// TwinCAT 3 PLC project Untitled1
// ProgramVersion: 3.1.4024.0
// libraries:
//   Tc2_Standard, * (Beckhoff Automation GmbH)
//   Tc2_System, * (Beckhoff Automation GmbH)
//   Tc2_Utilities, * (Beckhoff Automation GmbH)
//   Tc3_Module, * (Beckhoff Automation GmbH)
// project tree:
//   DUTs/ E_EventType.TcDUT, ST_Event.TcDUT (not stored)
//   / PlcTask.TcTTO
//   POUs/ FB_EventBuffer.TcPOU (not stored), MAIN.TcPOU (not stored)
// real-time tasks:
//   TASK PlcTask: cycle T#10ms, priority 20, ADS port 350

CONFIGURATION Untitled1
    RESOURCE PLC ON TwinCAT3
        TASK PlcTask(INTERVAL := T#10ms, PRIORITY := 20);
        PROGRAM MAIN WITH PlcTask : MAIN;
    END_RESOURCE
END_CONFIGURATION

// ---- DUTs/E_EventType.TcDUT
{attribute 'qualified_only'}
{attribute 'strict'}
TYPE E_EventType :
(
	Alarm := 0,
	Message := 1
);
END_TYPE
